Fanuc KAREL source: kt00252.KL

-- PROVISIONAL review KL for V1013-1; original PC SHA256 7666215b71671a5b68ab7b2cfffbae82ba342c18501d13a4c00f1b69854b3b2a
-- Incomplete behavior may be omitted. Consult companion uncertainty JSON. Do not deploy.
PROGRAM KT00252
%NOLOCKGROUP
VAR
  I2 : INTEGER
  OUT : INTEGER
-- UNRESOLVED_DECL H1 type=002017
BEGIN
  -- UNRESOLVED_PC offsets 5-19; opcodes 2E,22,9D,33,B4
  -- UNRESOLVED_PC offsets 24-35; opcodes 2E,23
  -- UNRESOLVED_PC offsets 40-62; opcodes 22,9D,33,B3,21,47,23
  -- UNRESOLVED_PC offsets 67-71; opcodes 7F
END KT00252
